Yaskawa INFORM job: PENDOWN.JBI

/JOB
//NAME PENDOWN
//POS
///NPOS 88,0,0,0,0,0
///TOOL 0
///POSTYPE PULSE
///PULSE
C00000=-2822,58859,-1118,-1041,-34109,-89
C00001=-2445,58590,-1551,-1095,-33918,-237
C00002=-2449,58587,-1561,-1095,-33912,-235
C00003=-2056,58784,-1255,-1143,-34035,-396
C00004=-1790,58767,-1273,-1178,-34027,-503
C00005=-1710,58665,-1427,-1190,-33965,-534
C00006=-1405,58500,-1671,-1233,-33866,-654
C00007=-1401,58503,-1661,-1233,-33872,-656
C00008=-1893,58484,-1701,-1169,-33857,-458
C00009=-1897,58481,-1711,-1169,-33851,-456
C00010=-1612,58342,-1916,-1209,-33767,-568
C00011=-1608,58345,-1906,-1209,-33773,-570
C00012=-1360,58476,-1701,-1239,-33856,-672
C00013=-1364,58473,-1711,-1239,-33850,-670
C00014=-1223,58270,-2017,-1261,-33725,-724
C00015=-1219,58273,-2007,-1261,-33731,-726
C00016=-2697,58359,-1905,-1065,-33776,-133
C00017=-2701,58356,-1915,-1065,-33770,-131
C00018=-2553,58520,-1665,-1082,-33870,-192
C00019=-2549,58523,-1655,-1082,-33876,-194
C00020=-1632,58127,-2238,-1209,-33639,-558
C00021=-1636,58124,-2248,-1209,-33633,-556
C00022=-1593,58292,-1992,-1212,-33736,-576
C00023=-1589,58295,-1982,-1212,-33742,-578
C00024=-1159,58148,-2197,-1271,-33654,-748
C00025=-1163,58145,-2207,-1271,-33648,-746
C00026=-1064,57873,-2621,-1289,-33479,-782
C00027=-1060,57876,-2611,-1289,-33485,-784
C00028=-2668,57792,-2760,-1078,-33433,-138
C00029=-2672,57789,-2770,-1078,-33427,-136
C00030=-2565,57980,-2481,-1089,-33542,-181
C00031=-2421,57972,-2491,-1108,-33538,-239
C00032=-2381,57921,-2568,-1114,-33507,-254
C00033=-2318,57966,-2498,-1122,-33534,-280
C00034=-2314,57969,-2488,-1122,-33540,-282
C00035=-1866,57724,-2852,-1185,-33391,-459
C00036=-1870,57721,-2862,-1185,-33385,-457
C00037=-1663,57735,-2839,-1212,-33393,-540
C00038=-1659,57738,-2829,-1212,-33399,-542
C00039=-2825,57234,-3603,-1065,-33095,-69
C00040=-2829,57231,-3613,-1065,-33089,-67
C00041=-2886,57431,-3312,-1054,-33210,-46
C00042=-2875,57923,-2571,-1049,-33508,-56
C00043=-2722,58308,-1988,-1063,-33741,-122
C00044=-2718,58311,-1978,-1063,-33747,-124
C00045=-1062,57706,-2870,-1292,-33380,-780
C00046=-1066,57703,-2880,-1292,-33374,-778
C00047=-1069,57484,-3214,-1296,-33238,-774
C00048=-1065,57487,-3204,-1296,-33244,-776
C00049=-2055,57490,-3210,-1164,-33248,-380
C00050=-2059,57487,-3220,-1164,-33242,-378
C00051=-2015,57631,-3001,-1167,-33330,-397
C00052=-1911,57724,-2860,-1180,-33387,-440
C00053=-1907,57727,-2850,-1180,-33393,-442
C00054=-1788,57452,-3266,-1200,-33224,-486
C00055=-1792,57449,-3276,-1200,-33218,-484
C00056=-1751,57398,-3352,-1206,-33186,-500
C00057=-1606,57439,-3288,-1225,-33211,-558
C00058=-1602,57442,-3278,-1225,-33217,-560
C00059=-1195,57081,-3825,-1286,-32993,-718
C00060=-1199,57078,-3835,-1286,-32987,-716
C00061=-1071,57339,-3436,-1298,-33148,-771
C00062=-1067,57342,-3426,-1298,-33154,-773
C00063=-2597,57248,-3581,-1095,-33102,-160
C00064=-2601,57245,-3591,-1095,-33096,-158
C00065=-2218,56760,-4322,-1154,-32798,-305
C00066=-2052,56777,-4296,-1176,-32807,-371
C00067=-1883,56965,-4011,-1196,-32921,-441
C00068=-1839,57109,-3791,-1199,-33009,-461
C00069=-1900,57185,-3676,-1190,-33057,-437
C00070=-2232,57104,-3802,-1147,-33008,-304
C00071=-2376,57135,-3755,-1127,-33028,-246
C00072=-2273,57106,-3799,-1141,-33010,-287
C00073=-1900,57185,-3676,-1190,-33057,-437
C00074=-1896,57188,-3666,-1190,-33063,-439
C00075=-1553,56660,-4468,-1245,-32735,-569
C00076=-1557,56657,-4478,-1245,-32729,-567
C00077=-1220,57030,-3907,-1284,-32957,-707
C00078=-1216,57033,-3897,-1284,-32963,-709
C00079=-2746,57034,-3905,-1078,-32973,-97
C00080=-2750,57031,-3915,-1078,-32967,-95
C00081=-2529,56725,-4375,-1113,-32780,-180
C00082=-2525,56728,-4365,-1113,-32786,-182
C00083=-2443,56676,-4445,-1125,-32753,-214
C00084=-2447,56673,-4455,-1125,-32747,-212
C00085=-2057,56484,-4741,-1181,-32628,-365
C00086=-1724,56567,-4615,-1224,-32675,-499
C00087=-1720,56570,-4605,-1224,-32681,-501
//INST
///DATE 2026/04/22 14:35
///ATTR SC,RW
///GROUP1 RB1
NOP
MOVJ C00000 VJ=0.78
MOVJ C00001 VJ=0.78
MOVJ C00002 VJ=0.78
MOVL C00003 V=20.0
MOVL C00004 V=20.0
MOVL C00005 V=20.0
MOVL C00006 V=20.0
MOVJ C00007 VJ=0.78
MOVJ C00008 VJ=0.78
MOVJ C00009 VJ=0.78
MOVL C00010 V=20.0
MOVJ C00011 VJ=0.78
MOVJ C00012 VJ=0.78
MOVJ C00013 VJ=0.78
MOVL C00014 V=20.0
MOVJ C00015 VJ=0.78
MOVJ C00016 VJ=0.78
MOVJ C00017 VJ=0.78
MOVL C00018 V=20.0
MOVJ C00019 VJ=0.78
MOVJ C00020 VJ=0.78
MOVJ C00021 VJ=0.78
MOVL C00022 V=20.0
MOVJ C00023 VJ=0.78
MOVJ C00024 VJ=0.78
MOVJ C00025 VJ=0.78
MOVL C00026 V=20.0
MOVJ C00027 VJ=0.78
MOVJ C00028 VJ=0.78
MOVJ C00029 VJ=0.78
MOVL C00030 V=20.0
MOVL C00031 V=20.0
MOVL C00032 V=20.0
MOVL C00033 V=20.0
MOVJ C00034 VJ=0.78
MOVJ C00035 VJ=0.78
MOVJ C00036 VJ=0.78
MOVL C00037 V=20.0
MOVJ C00038 VJ=0.78
MOVJ C00039 VJ=0.78
MOVJ C00040 VJ=0.78
MOVL C00041 V=20.0
MOVL C00042 V=20.0
MOVL C00043 V=20.0
MOVJ C00044 VJ=0.78
MOVJ C00045 VJ=0.78
MOVJ C00046 VJ=0.78
MOVL C00047 V=20.0
MOVJ C00048 VJ=0.78
MOVJ C00049 VJ=0.78
MOVJ C00050 VJ=0.78
MOVL C00051 V=20.0
MOVL C00052 V=20.0
MOVJ C00053 VJ=0.78
MOVJ C00054 VJ=0.78
MOVJ C00055 VJ=0.78
MOVL C00056 V=20.0
MOVL C00057 V=20.0
MOVJ C00058 VJ=0.78
MOVJ C00059 VJ=0.78
MOVJ C00060 VJ=0.78
MOVL C00061 V=20.0
MOVJ C00062 VJ=0.78
MOVJ C00063 VJ=0.78
MOVJ C00064 VJ=0.78
MOVL C00065 V=20.0
MOVL C00066 V=20.0
MOVL C00067 V=20.0
MOVL C00068 V=20.0
MOVL C00069 V=20.0
MOVL C00070 V=20.0
MOVL C00071 V=20.0
MOVL C00072 V=20.0
MOVL C00073 V=20.0
MOVJ C00074 VJ=0.78
MOVJ C00075 VJ=0.78
MOVJ C00076 VJ=0.78
MOVL C00077 V=20.0
MOVJ C00078 VJ=0.78
MOVJ C00079 VJ=0.78
MOVJ C00080 VJ=0.78
MOVL C00081 V=20.0
MOVJ C00082 VJ=0.78
MOVJ C00083 VJ=0.78
MOVJ C00084 VJ=0.78
MOVL C00085 V=20.0
MOVL C00086 V=20.0
MOVJ C00087 VJ=0.78
END
